(* CoDeSys 2.3.9.62 project: Cap5_ej1.pro *)
(* Libraries: Standard.lib 4.10.05 10:14:46, IecSfc.lib*2.6.14 10:37:46 *)

(* POU PLC_PRG, FBD *)
PROGRAM PLC_PRG
VAR

   BotonS : BOOL;
   BotonR : BOOL;
   Salida: BOOL;
   MiBiestable : Biestable;

END_VAR
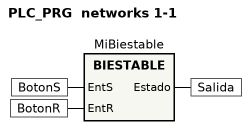
_FBD_ (* Function Block Diagram *)
NETWORK 1
	MiBiestable:BIESTABLE(EntS: BotonS, EntR: BotonR) => Salida
_END_FBD_
(* the same logic as Structured Text *)
(* Network 1 *)
MiBiestable(EntS := BotonS, EntR := BotonR);
Salida := MiBiestable.Estado;
END_PROGRAM

(* POU Biestable, ST *)
FUNCTION_BLOCK Biestable
VAR_INPUT
   EntS : BOOL;
   EntR:BOOL;
END_VAR
VAR_OUTPUT
    Estado : BOOL := FALSE;
END_VAR
VAR
END_VAR
IF (EntS=TRUE ) THEN
   Estado:=TRUE;
ELSE
   IF (EntR=TRUE) THEN
       Estado:=FALSE;
   END_IF
END_IF
END_FUNCTION_BLOCK

(* Visualisation Biestable
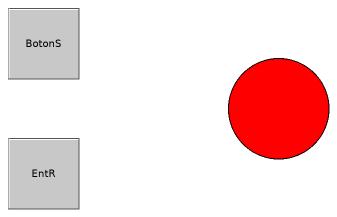
button at (110,80)-(181,151): text "BotonS"; taps PLC_PRG.BotonS
button at (110,210)-(181,281): text "EntR"; taps PLC_PRG.BotonR
ellipse at (330,130)-(431,231): alarm colour if PLC_PRG.Salida
*)
